RoboDK station: Stringer B-Corner-Bot-Short-BOX2.rdk

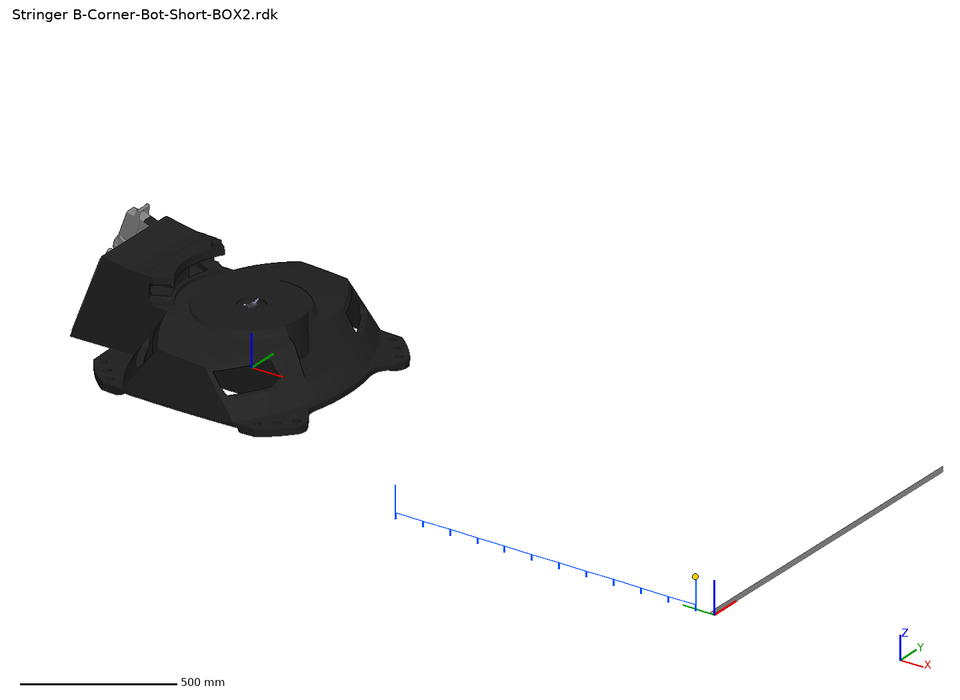
[picture v0: the station drawn from its stored meshes, robots at their saved joint values, targets as dots, program paths as lines]
Station Stringer B-Corner-Bot-Short-BOX2 (saved by RoboDK 5.2.3). Poses are relative to the parent item; angles as X-Y-Z fixed-axis rotations.
  - frame KUKA KR 210 R2700 extra Base at (0, 0, 0) mm
    - robot KUKA KR 210 R2700 extra: 6 axes, payload 210 kg, reach 2696 mm, repeatability 0.06 mm, weight 1068 kg
        joint limits [-185, -140, -120, -350, -125, -350] to [185, -5, 155, 350, 125, 350]; home [0, -90, 90, 0, 0, 0]; saved at [-39.117, -26.624, 86.023, 93.553, 23.441, -126.163]
      - tool Spindle, TCP at (32, 0, 260) mm, rotated rx 0 ry 39 rz 0 deg, size 157.3 x 72 x 259.9 mm
  - frame Frame 2 at (1800, 0, -372.68) mm, rotated rx 0 ry 0 rz 90 deg
    - object Stringer B-Corner-Bot-Short-BOX2 at (0, 0, 0) mm, rotated rx 0 ry 0 rz -90 deg, 12 curves, geometry from Point 12
    - object L-Stringer B-bottom-short-corner - box2 at (0, 0, 0) mm, size 1281.1 x 20 x 20 mm, geometry from L-Stringer B-bottom-short-corner - box2.stl
  - machining project Point settings: rotZ(0) | rotX(0)*rotY(0) | rotz(0) | onStart | onPathStart | onApproach | onPoint | onRetract | onFinish | SetRPM(%1) | SetTool(%1) | Extruder(%1) | default | default | OutOnMov(%1) | OutOffMov(%1) | onPathFinish | M_RunCode(%1) | riverData=C:\Windows\System32\Driv | PS_BROWSER_APP_PROFILE_STRING=Inter | PS_BROWSER_USER_PROFILE_STRING=Defa | OCALAPPDATA=C:\Users\jbert\AppData\Loc | OneDrive=C:\Users\jbert\O | Path=C:\Program Files (x86)\NVIDIA Corpora
  - program Point (71 instructions, listed below)
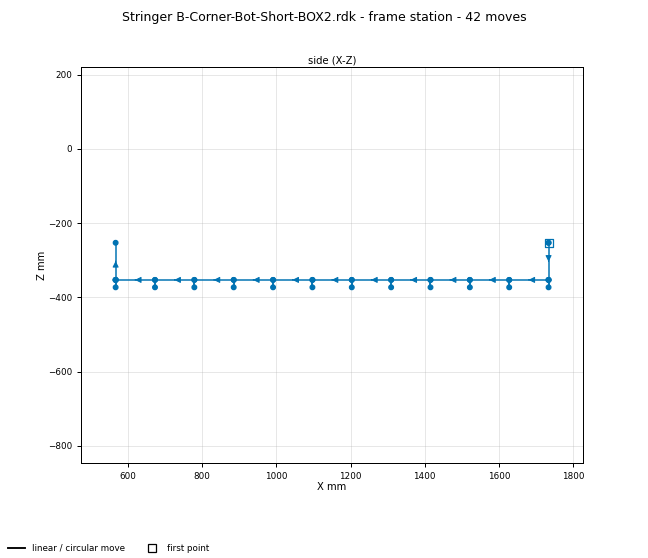
[picture p0: tool path of Stringer B-Corner-Bot-Short-BOX2.rdk in frame station, 42 of 42 moves have a stored position in this frame; points joined in program order, loops and branches not executed]

--- program Point (robot KUKA KR 210 R2700 extra) ---
  Smooth(1)
  Set speed (1000.0 mm/s)
  Set Ref.: Frame 2
  Set Tool: Spindle
  Show Spindle
  MoveJ 1 to (-10.2, 66.57, 120) mm, rotated rx -180 ry 0 rz -180 deg; joints [-2.515, -34.002, 111.787, 176.489, 26.801, -178.82]
  MoveL 2 to (-10.2, 66.57, 120) mm, rotated rx -180 ry 0 rz -180 deg; joints [-2.515, -34.002, 111.787, 176.489, 26.801, -178.82]
  MoveL 3 to (-10.2, 66.57, 20) mm, rotated rx 180 ry 0 rz 180 deg; joints [-2.515, -28.676, 109.145, 176.784, 29.481, -179.154]
  MoveL 4 to (-10.2, 66.57, 20) mm, rotated rx 180 ry 0 rz 180 deg; joints [-2.515, -28.676, 109.145, 176.784, 29.481, -179.154]
  Set speed (50.0 mm/s)
  MoveL 5 to (-10.2, 66.57, 0) mm, rotated rx 180 ry 0 rz 180 deg; joints [-2.515, -27.618, 108.57, 176.831, 29.962, -179.208]
  MoveL 6 to (-10.2, 66.57, 20) mm, rotated rx 180 ry 0 rz 180 deg; joints [-2.515, -28.676, 109.145, 176.784, 29.481, -179.154]
  Set speed (1000.0 mm/s)
  MoveL 7 to (-10.2, 172.57, 20) mm, rotated rx -180 ry 0 rz -180 deg; joints [-6.495, -28.616, 108.712, 171.604, 29.178, -177.713]
  Set speed (50.0 mm/s)
  MoveL 8 to (-10.2, 172.57, 0) mm, rotated rx 180 ry 0 rz 180 deg; joints [-6.495, -27.562, 108.138, 171.727, 29.652, -177.854]
  MoveL 9 to (-10.2, 172.57, 20) mm, rotated rx -180 ry 0 rz -180 deg; joints [-6.495, -28.616, 108.712, 171.604, 29.178, -177.713]
  Set speed (1000.0 mm/s)
  MoveL 10 to (-10.2, 278.57, 20) mm, rotated rx 180 ry 0 rz 180 deg; joints [-10.414, -28.496, 107.896, 166.266, 28.628, -176.02]
  Set speed (50.0 mm/s)
  MoveL 11 to (-10.2, 278.57, 0) mm, rotated rx -180 ry 0 rz -180 deg; joints [-10.414, -27.45, 107.325, 166.469, 29.09, -176.252]
  MoveL 12 to (-10.2, 278.57, 20) mm, rotated rx 180 ry 0 rz 180 deg; joints [-10.414, -28.496, 107.896, 166.266, 28.628, -176.02]
  Set speed (1000.0 mm/s)
  MoveL 13 to (-10.2, 384.57, 20) mm, rotated rx 180 ry 0 rz 180 deg; joints [-14.237, -28.306, 106.699, 160.668, 27.873, -173.925]
  Set speed (50.0 mm/s)
  MoveL 14 to (-10.2, 384.57, 0) mm, rotated rx -180 ry 0 rz -180 deg; joints [-14.237, -27.27, 106.132, 160.957, 28.316, -174.252]
  MoveL 15 to (-10.2, 384.57, 20) mm, rotated rx 180 ry 0 rz 180 deg; joints [-14.237, -28.306, 106.699, 160.668, 27.873, -173.925]
  Set speed (1000.0 mm/s)
  MoveL 16 to (-10.2, 490.57, 20) mm, rotated rx -180 ry 0 rz -180 deg; joints [-17.934, -28.031, 105.125, 154.705, 26.97, -171.278]
  Set speed (50.0 mm/s)
  MoveL 17 to (-10.2, 490.57, 0) mm, rotated rx -180 ry 0 rz -180 deg; joints [-17.934, -27.008, 104.563, 155.086, 27.387, -171.706]
  MoveL 18 to (-10.2, 490.57, 20) mm, rotated rx -180 ry 0 rz -180 deg; joints [-17.934, -28.031, 105.125, 154.705, 26.97, -171.278]
  Set speed (1000.0 mm/s)
  MoveL 19 to (-10.2, 596.57, 20) mm, rotated rx 180 ry 0 rz 180 deg; joints [-21.484, -27.654, 103.177, 148.269, 25.991, -167.941]
  Set speed (50.0 mm/s)
  MoveL 20 to (-10.2, 596.57, 0) mm, rotated rx 180 ry 0 rz 180 deg; joints [-21.484, -26.647, 102.621, 148.748, 26.375, -168.475]
  MoveL 21 to (-10.2, 596.57, 20) mm, rotated rx 180 ry 0 rz 180 deg; joints [-21.484, -27.654, 103.177, 148.269, 25.991, -167.941]
  Set speed (1000.0 mm/s)
  MoveL 22 to (-10.2, 702.57, 20) mm, rotated rx 180 ry 0 rz 180 deg; joints [-24.868, -27.156, 100.858, 141.264, 25.021, -163.797]
  Set speed (50.0 mm/s)
  MoveL 23 to (-10.2, 702.57, 0) mm, rotated rx 180 ry 0 rz -180 deg; joints [-24.868, -26.166, 100.306, 141.844, 25.365, -164.438]
  MoveL 24 to (-10.2, 702.57, 20) mm, rotated rx 180 ry 0 rz 180 deg; joints [-24.868, -27.156, 100.858, 141.264, 25.021, -163.797]
  Set speed (1000.0 mm/s)
  MoveL 25 to (-10.2, 808.57, 20) mm, rotated rx 180 ry 0 rz -180 deg; joints [-28.078, -26.519, 98.167, 133.626, 24.154, -158.767]
  Set speed (50.0 mm/s)
  MoveL 26 to (-10.2, 808.57, 0) mm, rotated rx 180 ry 0 rz 180 deg; joints [-28.078, -25.548, 97.621, 134.303, 24.449, -159.51]
  MoveL 27 to (-10.2, 808.57, 20) mm, rotated rx 180 ry 0 rz -180 deg; joints [-28.078, -26.519, 98.167, 133.626, 24.154, -158.767]
  Set speed (1000.0 mm/s)
  MoveL 28 to (-10.2, 914.57, 20) mm, rotated rx 180 ry 0 rz 180 deg; joints [-31.106, -25.725, 95.103, 125.347, 23.491, -152.84]
  Set speed (50.0 mm/s)
  MoveL 29 to (-10.2, 914.57, 0) mm, rotated rx 180 ry 0 rz -180 deg; joints [-31.106, -24.773, 94.561, 126.109, 23.73, -153.671]
  MoveL 30 to (-10.2, 914.57, 20) mm, rotated rx 180 ry 0 rz 180 deg; joints [-31.106, -25.725, 95.103, 125.347, 23.491, -152.84]
  Set speed (1000.0 mm/s)
  MoveL 31 to (-10.2, 1020.57, 20) mm, rotated rx 180 ry 0 rz -180 deg; joints [-33.953, -24.753, 91.66, 116.516, 23.129, -146.103]
  Set speed (50.0 mm/s)
  MoveL 32 to (-10.2, 1020.57, 0) mm, rotated rx -180 ry 0 rz -180 deg; joints [-33.953, -23.821, 91.121, 117.333, 23.307, -146.992]
  MoveL 33 to (-10.2, 1020.57, 20) mm, rotated rx 180 ry 0 rz -180 deg; joints [-33.953, -24.753, 91.66, 116.516, 23.129, -146.103]
  Set speed (1000.0 mm/s)
  MoveL 34 to (-10.2, 1126.57, 20) mm, rotated rx 180 ry 0 rz -180 deg; joints [-36.621, -23.586, 87.825, 107.327, 23.157, -138.754]
  Set speed (50.0 mm/s)
  MoveL 35 to (-10.2, 1126.57, 0) mm, rotated rx -180 ry 0 rz -180 deg; joints [-36.621, -22.673, 87.287, 108.16, 23.271, -139.66]
  MoveL 36 to (-10.2, 1126.57, 20) mm, rotated rx 180 ry 0 rz -180 deg; joints [-36.621, -23.586, 87.825, 107.327, 23.157, -138.754]
  Set speed (1000.0 mm/s)
  MoveL 37 to (-10.2, 1232.57, 20) mm, rotated rx -180 ry 0 rz -180 deg; joints [-39.117, -22.203, 83.577, 98.066, 23.641, -131.085]
  Set speed (50.0 mm/s)
  MoveL 38 to (-10.2, 1232.57, 0) mm, rotated rx 180 ry 0 rz -180 deg; joints [-39.117, -21.308, 83.037, 98.867, 23.694, -131.96]
  MoveL 39 to (-10.2, 1232.57, 20) mm, rotated rx -180 ry 0 rz -180 deg; joints [-39.117, -22.203, 83.577, 98.066, 23.641, -131.085]
  MoveL 40 to (-10.2, 1232.57, 20) mm, rotated rx -180 ry 0 rz -180 deg; joints [-39.117, -22.203, 83.577, 98.066, 23.641, -131.085]
  Set speed (1000.0 mm/s)
  MoveL 41 to (-10.2, 1232.57, 20) mm, rotated rx -180 ry 0 rz -180 deg; joints [-39.117, -22.203, 83.577, 98.066, 23.641, -131.085]
  MoveL 42 to (-10.2, 1232.57, 120) mm, rotated rx -180 ry 0 rz -180 deg; joints [-39.117, -26.624, 86.023, 93.553, 23.441, -126.163]
